(* IEC 61131-3 sources: HappyLearnCodesys/content/softmotion/Robotics_PickAndPlace, 6 files *)

(* ---- GVL.st ---- *)
(*
    檔案用途：定義本範例中三角機器人、輸送帶與旋轉工作台的幾何位置常數，
              以及用來切換「自動／手動放環」的全域旗標。
    教學重點：這些數值會直接影響實際運動軌跡與畫面位置，修改前請先對照
              `DeviceTree_Axes.md` 與各 POU 程式中的使用方式再調整。
*)
VAR_GLOBAL CONSTANT
    gcTripodTransX : LREAL := 0;       // Tripod 機構在世界座標中的 X 平移量
    gcTripodTransY : LREAL := 0;       // Tripod 機構在世界座標中的 Y 平移量
    gcTripodTransZ : LREAL := 1700;    // Tripod 機構在世界座標中的 Z 平移量（機器人高度）

    gcTripodSize : LREAL := 180;       // Tripod 幾何尺寸基準，影響工作空間與 TCP 半徑

    gcBeltTransX : LREAL := 0;         // 輸送帶座標系（PCS_2）在世界座標中的 X 位置
    gcBeltTransY : LREAL := 500;       // 輸送帶座標系在世界座標中的 Y 位置
    gcBeltTransZ : LREAL := 0;         // 輸送帶座標系在世界座標中的 Z 位置

    gcTableTransX : LREAL := 0;        // 旋轉工作台座標系（PCS_1）在世界座標中的 X 位置
    gcTableTransY : LREAL := -500;     // 旋轉工作台座標系在世界座標中的 Y 位置
    gcTableTransZ : LREAL := 0;        // 旋轉工作台座標系在世界座標中的 Z 位置

    gcTCP_Ring : LREAL := 0.02 * gcTripodSize + 15;   // 末端工具座標系到圓環下緣的距離

    gcTripod1PosOrig : LREAL := 50;    // Tripod1 初始軸位置
    gcTripod2PosOrig : LREAL := 75;    // Tripod2 初始軸位置
    gcTripod3PosOrig : LREAL := 25;    // Tripod3 初始軸位置
END_VAR
VAR_GLOBAL
    gbSetRing : BOOL;                  // TRUE：由操作者手動要求在轉盤上放一個新環
    gbAutomatic : BOOL := TRUE;        // TRUE：環依邏輯自動連續產生；FALSE：完全由 gbSetRing 控制
END_VAR

(* ---- Cone.st ---- *)
(*
    檔案用途：
      以狀態機方式描述單一圓錐（Cone）在輸送帶上的一生：
      何時出現、如何被輸送帶帶動、何時離開工作區域，以及如何更新 PCS_2。
    教學重點：
      - 透過 MC_TrackConveyorBelt 追蹤輸送帶上的物件位置，並與 Tripod 軸組連動。
      - 觀察 REPEAT / UNTIL 與 state / stateOld 的組合，如何實作「直到狀態穩定」的迴圈。
      - 理解 pActiveCone 與 pPreviousCone 指標，如何在三顆圓錐之間接續產生與移動。
*)
FUNCTION_BLOCK Cone
VAR_IN_OUT
	pActiveCone : POINTER TO Cone;
END_VAR
VAR_INPUT
	pPreviousCone : POINTER TO Cone;
END_VAR
VAR_OUTPUT
	pos : MC_COORD_REF;
	state : DINT;
	bOnBelt : BOOL;
END_VAR
VAR
	conveyorBeltOrigin : MC_COORD_REF := (X := gcBeltTransX, Y := gcBeltTransY, Z := gcBeltTransZ);
	initialConePosition : MC_COORD_REF := (X := -925, Z := 125);
	tcb : MC_TrackConveyorBelt := (ConveyorBeltOrigin := conveyorBeltOrigin,
								   InitialObjectPosition := initialConePosition,
								   CoordSystem := SMC_COORD_SYSTEM.PCS_2);
	f : SMC_Frame;
	stateOld : DINT;
END_VAR

REPEAT
	stateOld := state;
	CASE state OF
	0:	//cone invisible
		IF NOT Robot.bDontChangePCS_2 THEN
			IF pPreviousCone^.bOnBelt AND pPreviousCone^.pos.X >= -250 THEN
				tcb(Execute := FALSE, AxisGroup := Tripod, ConveyorBelt := DriveConveyorBelt);
				tcb.Execute := TRUE;
				state := state + 10;
			END_IF
		END_IF
	10:	//linking PCS_2 to the position of the cone
		IF tcb.Done THEN
			bOnBelt := TRUE;
			pActiveCone := THIS;
			state := state + 10;
		END_IF
	20:	//cone on belt
		tcb.cs.GetPose(cs := f, fTime := Tripod1.fTaskCycle);
		SMC_Frame_To_CoordRef(c := pos, f := f);
		IF pos.X >= gcBeltTransX + 725 THEN
			bOnBelt := FALSE;
			state := 0;
		END_IF
	END_CASE
	tcb(AxisGroup := Tripod, ConveyorBelt := DriveConveyorBelt);
UNTIL state = stateOld
END_REPEAT

(* ---- Ring.st ---- *)
(*
    檔案用途：
      以狀態機方式描述單一圓環（Ring）從轉盤待命、被機器人取走、
      一直到被放到圓錐上、再回到初始狀態的整個流程。
    教學重點：
      - 使用 MC_TrackRotaryTable 取得轉盤上物件的即時位置，並映射到 PCS_1。
      - 觀察如何根據 Robot 的輸出旗標（bReadyForMotion、bRingAttached、pTargetCone）
        來協調「轉盤上兩個圓環」與「機器人」之間的合作。
      - 練習閱讀以 DINT state 切分的多段狀態（0/10/20/30/40/50），對照實際動作想像流程。
*)
FUNCTION_BLOCK Ring
VAR_INPUT
	pOtherRing : POINTER TO Ring;
	startPos : MC_COORD_REF;
END_VAR
VAR_OUTPUT
	pos : MC_COORD_REF;
	state : DINT;
	bOnTable : BOOL;
END_VAR
VAR
	stateOld : DINT;
	fTemp : LREAL;
	f : SMC_Frame;
	rotaryTableOrigin : MC_COORD_REF := (X := gcTableTransX, Y := gcTableTransY, Z := gcTableTransZ);
	initialObjectPosition : MC_COORD_REF := (Y := 400, Z := 20 + 10);
	trt : MC_TrackRotaryTable := (RotaryTableOrigin := rotaryTableOrigin, initialObjectPosition := initialObjectPosition, CoordSystem := SMC_COORD_SYSTEM.PCS_1);
	pCone : POINTER TO Cone;
END_VAR

REPEAT
	stateOld := state;
	CASE state OF
	0:	//ring at original position
		pos := startPos;
		IF Robot.bReadyForMotion AND
		   (pOtherRing^.state = 0 OR pOtherRing^.state >= 40) AND
		   (gbSetRing OR gbAutomatic) THEN
			trt(Execute := FALSE, AxisGroup := Tripod, RotaryTable := DriveRotaryTable);
			trt.Execute := TRUE;
			state := state + 10;
		END_IF

	10:	//linking PCS_1 to the position of the ring
		IF trt.Done THEN
			state := state + 10;
		END_IF

	20:	//ring on rotary-table, wait until robot is free
		trt.cs.GetPose(cs := f, fTime := Tripod1.fTaskCycle);
		SMC_Frame_To_CoordRef(c := pos, f := f);
		IF NOT Robot.bRingAttached THEN
			state := state + 10;
		END_IF

	30: //waiting for takeoff
		trt.cs.GetPose(cs := f, fTime := Tripod1.fTaskCycle);
		SMC_Frame_To_CoordRef(c := pos, f := f);
		IF Robot.bRingAttached THEN
			state := state + 10;
		END_IF

	40:	//ring attached to robot
		pos.X := Robot.readPos.Position.c.X;
		pos.Y := Robot.readPos.Position.c.Y;
		pos.Z := Robot.readPos.Position.c.Z - gcTCP_Ring;
		IF NOT Robot.bRingAttached THEN
			pCone := Robot.pTargetCone;
			state := state + 10;
		END_IF

	50:	//ring placed on cone
		pos.X := pCone^.pos.X;
		pos.Y := pCone^.pos.Y;
		pos.Z := pCone^.pos.Z;
		IF NOT pCone^.bOnBelt THEN
			state := 0;
		END_IF
	END_CASE

	trt(AxisGroup := Tripod, RotaryTable := DriveRotaryTable);
UNTIL state = stateOld
END_REPEAT

bOnTable := state = 20 OR state = 30;

(* ---- DepictorCalculations.st ---- *)
(*
    檔案用途：
      計算用於可視化的標記座標陣列 aafPos，讓視覺介面能畫出輸送帶路徑
      以及 Tripod 運動軌跡的參考線。
    教學重點：
      - 透過 Tripod_Lin_Depictor 取得 Tripod 軸組的線性插補資訊，作為可視化基底。
      - 使用 SIN、COS 與多段 if/else 邏輯，組合出一條封閉的輸送帶路徑。
      - 練習將實際軸位置（DriveConveyorBelt.fSetPosition 等）轉換成畫面上的座標點。
*)
PROGRAM DepictorCalculations
VAR_OUTPUT
	aafPos : ARRAY[0..9] OF ARRAY[0..1] OF LREAL;
END_VAR
VAR
	dep : Tripod_Lin_Depictor;
	fTemp : LREAL;
	i : INT;
END_VAR

//tripod
IF Robot.state >= 40 THEN
	dep(group := Tripod, kin := Tripod.trafo);
END_IF

//markings on belt
FOR i := 0 TO 9 DO
	fTemp := DriveConveyorBelt.fSetPosition + INT_TO_LREAL(i) / 10 * DriveConveyorBelt.fPositionPeriod;
	IF fTemp >= DriveConveyorBelt.fPositionPeriod THEN
		fTemp := fTemp - DriveConveyorBelt.fPositionPeriod;
	END_IF

	IF fTemp <= 1000 THEN
		aafPos[i][0] := fTemp;
		aafPos[i][1] := 50;
	ELSE
		fTemp := fTemp - 1000;
		IF fTemp < 50 * SMC_PI THEN
			aafPos[i][0] := 1000 + 50 * SIN(fTemp / 50);
			aafPos[i][1] := 50 * COS(fTemp / 50);
		ELSE
			fTemp := fTemp - 50 * SMC_PI;
			IF fTemp <= 2000 THEN
				aafPos[i][0] := 1000 - fTemp;
				aafPos[i][1] := -50;
			ELSE
				fTemp := fTemp - 2000;
				IF fTemp < 50 * SMC_PI THEN
					aafPos[i][0] := -1000 - 50 * SIN(fTemp / 50);
					aafPos[i][1] := -50 * COS(fTemp / 50);
				ELSE
					fTemp := fTemp - 50 * SMC_PI;
					aafPos[i][0] := -1000 + fTemp;
					aafPos[i][1] := 50;
				END_IF
			END_IF
		END_IF
	END_IF
END_FOR

(* ---- Environment.st ---- *)
(*
    檔案用途：
      負責「環境」相關的裝置控制，包括旋轉工作台與輸送帶的驅動，
      並管理所有圓錐（Cone）與圓環（Ring）的狀態機，提供給機器人程式使用。
    教學重點：
      - 將與機器人本體無關、但會影響工作流程的設備集中在一支 PROGRAM 中管理。
      - 觀察如何透過 FUNCTION_BLOCK 實例（Cone、Ring）與指標，建立物件之間的關聯。
      - 使用簡單的初始化旗標 bInit 來區分「第一次循環」與「正常運轉」的寫法。
*)
PROGRAM Environment
VAR_OUTPUT
	cone1, cone2, cone3 : Cone;
	ring1, ring2 : Ring;
	bRingOnTable : BOOL;
	pActiveCone : POINTER TO Cone;	//the cone corresponding to PCS_2
END_VAR
VAR
	powRotaryTable : MC_Power := (Enable := TRUE, bRegulatorOn := TRUE, bDriveStart := TRUE);
	powConveyorBelt : MC_Power := (Enable := TRUE, bRegulatorOn := TRUE, bDriveStart := TRUE);
	mvRotaryTable : MC_MoveVelocity := (Execute := TRUE, Velocity := 50, Acceleration := 30, Deceleration := 30, Jerk := 1000);
	mvConveyorBelt : MC_MoveVelocity := (Execute := TRUE, Velocity := 300, Acceleration := 150, Deceleration := 150, Jerk := 1000);

	ring1StartPos : MC_COORD_REF := (X := 75, Y := 100, Z := 0);
	ring2StartPos : MC_COORD_REF := (X := -75, Y := 100, Z := 0);
	bInit : BOOL := TRUE;
END_VAR

//moving rotary-table-/ conveyor-belt-drive
powRotaryTable(Axis := DriveRotaryTable);
powConveyorBelt(Axis := DriveConveyorBelt);
IF NOT (powRotaryTable.Status AND powConveyorBelt.Status) THEN
	RETURN;
END_IF
mvRotaryTable(Axis := DriveRotaryTable);
mvConveyorBelt(Axis := DriveConveyorBelt);

//state-machines of cones / handling of PCS_2
IF bInit THEN
	cone1.Start();
END_IF
cone1(pActiveCone := pActiveCone, pPreviousCone := ADR(cone3));
cone2(pActiveCone := pActiveCone, pPreviousCone := ADR(cone1));
cone3(pActiveCone := pActiveCone, pPreviousCone := ADR(cone2));

//state-machines of rings / handling of PCS_1
IF bInit THEN
	ring1.startPos := ring1StartPos;
	ring2.startPos := ring2StartPos;
END_IF
ring1(pOtherRing := ADR(ring2));
ring2(pOtherRing := ADR(ring1));
bRingOnTable := ring1.bOnTable OR ring2.bOnTable;

bInit := FALSE;

(* ---- Robot.st ---- *)
(*
    檔案用途：
      控制 Tripod 三角機器人完成「從旋轉工作台拾取圓環，放置到輸送帶上圓錐」的
      完整 Pick & Place 循環，並回報目前是否可動作與是否已夾持圓環。
    教學重點：
      - 觀察如何使用多顆 MC_Power、MC_SetPosition、MC_MoveLinear* 等運動控制 FB
        來建立啟動流程與多段直線軌跡。
      - 搭配座標系（WCS、PCS_1、PCS_2）與位置常數，理解不同工位之間的轉換。
      - 透過整數變數 state 所構成的狀態機，練習閱讀與設計順序控制流程。
*)
PROGRAM Robot
VAR_OUTPUT
    bReadyForMotion : BOOL;
	bRingAttached : BOOL;
	bDontChangePCS_2 : BOOL;	//there are several commands using PCS_2, which shall not change in the meantime
	pTargetCone : POINTER TO Cone;
END_VAR
VAR
    pwA1 : MC_Power := (Enable:= TRUE, bRegulatorOn:= TRUE, bDriveStart:= TRUE);
    pwA2 : MC_Power := (Enable:= TRUE, bRegulatorOn:= TRUE, bDriveStart:= TRUE);
    pwA3 : MC_Power := (Enable:= TRUE, bRegulatorOn:= TRUE, bDriveStart:= TRUE);
    spA1, spA2, spA3 : MC_SetPosition;

	enable : MC_GroupEnable;
	setCoord : MC_SetCoordinateTransform;
    mcs : MC_COORD_REF;

    mvToRing : MC_MoveLinearAbsolute := (Velocity := VEL, Acceleration := ACC, Deceleration := ACC, Jerk := JRK, Name:= 'Move to ring');
	mvToRestPos : MC_MoveLinearAbsolute := (Velocity := VEL, Acceleration := ACC, Deceleration := ACC, Jerk := JRK, Name:= 'Move to rest position');
	mvAboveCone : MC_MoveLinearAbsolute := (Velocity := VEL, Acceleration := ACC, Deceleration := ACC, Jerk := JRK, Name:= 'Move above cone');
	mvUpFromRing : MC_MoveLinearRelative := (Velocity := VEL, Acceleration := ACC, Deceleration := ACC, Jerk := JRK, Name:= 'Move up from ring');

	mvDownToCone : MC_MoveLinearAbsolute := (Velocity := VEL, Acceleration := ACC, Deceleration := ACC, Jerk := JRK, Name:= 'Move down to cone');
	mvUpFromCone : MC_MoveLinearAbsolute := (Velocity := VEL, Acceleration := ACC, Deceleration := ACC, Jerk := JRK, Name:= 'Move up from cone');

    mvBack : MC_MoveLinearAbsolute := (Velocity := VEL, Acceleration := ACC, Deceleration := ACC, Jerk := JRK, Name:= 'Move back');

	readStatus : MC_GroupReadStatus;
    readPos : MC_GroupReadActualPosition;

	state : INT;
	ton : TON := (PT := T#200MS);
END_VAR
VAR CONSTANT
    VEL : LREAL :=   1000 ;
    ACC : LREAL :=  10000 ;
    JRK : LREAL := 100000 ;

    POS_ABOVE_RING_PCS_1 : SMC_POS_REF := (c:= (X:= 0, Y:= 0, Z:= gcTCP_Ring)) ;
    POS_ABOVE_CONE_PCS_2 : SMC_POS_REF := (c:= (X:= 0, Y:= 0, Z:= 200)) ;
    POS_ON_CONE_PCS_2 : SMC_POS_REF := (c:= (X:= 0, Y:= 0, Z:= gcTCP_Ring)) ;
    POS_REST_WCS : SMC_POS_REF := (c:= (X:= 0, Y:= 0, Z:= 300)) ;
END_VAR

pwA1(Axis:= Tripod1);
pwA2(Axis:= Tripod2);
pwA3(Axis:= Tripod3);

CASE state OF
0:
    IF pwA1.Status AND pwA2.Status AND pwA3.Status THEN
        state := state + 10;
	END_IF

10:	//starting at given axis-positions
    spA1(Axis:= Tripod1, Execute:= TRUE, Position:= gcTripod1PosOrig);
    spA2(Axis:= Tripod2, Execute:= TRUE, Position:= gcTripod2PosOrig);
    spA3(Axis:= Tripod3, Execute:= TRUE, Position:= gcTripod3PosOrig);

    IF spA1.Done AND spA2.Done AND spA3.Done THEN
		setCoord(AxisGroup := Tripod, Execute := FALSE);
        state := state + 10;
	END_IF

20:	//telling the robot its position in space
	mcs.X := gcTripodTransX;
	mcs.Y := gcTripodTransY;
	mcs.Z := gcTripodTransZ;
    setCoord(
	        AxisGroup := Tripod,
            Execute := TRUE,
            CoordTransform := mcs,
            CoordSystem := SMC_COORD_SYSTEM.MCS);

    IF setCoord.Done THEN
        state := state + 10;
	END_IF

30: //enabling the axis group
    enable(AxisGroup:= Tripod, Execute:= TRUE);
    IF enable.Done THEN
		state := state + 10;
    END_IF

40:
	IF Environment.bRingOnTable THEN
		//approaching a ring on the table
		mvToRing(AxisGroup:= Tripod, Execute := FALSE);
		mvToRing.Position := POS_ABOVE_RING_PCS_1 ;
		mvToRing.BufferMode := MC_BUFFER_MODE.BlendingHigh;
		mvToRing.TransitionMode := MC_TRANSITION_MODE.TMCornerDistance;
		mvToRing.TransitionParameter[0] := 500;
		mvToRing.CoordSystem := SMC_COORD_SYSTEM.PCS_1;
		mvToRing.Execute := TRUE;
    	state := state + 10;
	END_IF

50:
    IF mvToRing.Done THEN
		ton(IN := FALSE);
		state := state + 10;
	END_IF

60:
	ton(IN := TRUE);
	//waiting some time (following the ring)
	IF ton.Q THEN
		//moving upwards (still in PCS_1)
		mvUpFromRing(AxisGroup:= Tripod, Execute := FALSE);
		mvUpFromRing.Distance.c.Z := 150;
		mvUpFromRing.CoordSystem := SMC_COORD_SYSTEM.PCS_1;
		mvUpFromRing.BufferMode := MC_BUFFER_MODE.Buffered;
		mvUpFromRing.TransitionMode := MC_TRANSITION_MODE.TMNone;
		mvUpFromRing.Execute := TRUE;
		state := state + 10;
	END_IF

70:
	IF mvUpFromRing.CommandAccepted THEN
		//neutral position
		mvToRestPos(AxisGroup:= Tripod, Execute := FALSE);
		mvToRestPos.Position := POS_REST_WCS ;
		mvToRestPos.CoordSystem := SMC_COORD_SYSTEM.WCS;
		mvToRestPos.BufferMode := MC_BUFFER_MODE.BlendingHigh;
		mvToRestPos.TransitionMode := MC_TRANSITION_MODE.TMCornerDistance;
		mvToRestPos.TransitionParameter[0] := 500 ;
		mvToRestPos.Execute := TRUE;
		state := state + 10;
	END_IF

80:
	IF mvToRestPos.CommandAccepted THEN
		//moving to some position above the next cone
		pTargetCone := Environment.pActiveCone;
		mvAboveCone(AxisGroup:= Tripod, Execute := FALSE);
		mvAboveCone.Position := POS_ABOVE_CONE_PCS_2 ;
		mvAboveCone.CoordSystem := SMC_COORD_SYSTEM.PCS_2;
		mvAboveCone.BufferMode := MC_BUFFER_MODE.BlendingHigh;
		mvAboveCone.TransitionMode := MC_TRANSITION_MODE.TMCornerDistance;
        mvAboveCone.TransitionParameter[0] := 1000 ;
		mvAboveCone.Execute := TRUE;
		state := state + 10;
	END_IF

90:
	IF mvAboveCone.CommandAccepted THEN
		//approaching the cone
		mvDownToCone(AxisGroup:= Tripod, Execute := FALSE);
		mvDownToCone.Position := POS_ON_CONE_PCS_2 ;
		mvDownToCone.BufferMode := MC_BUFFER_MODE.BlendingHigh;
		mvDownToCone.TransitionMode := MC_TRANSITION_MODE.TMCornerDistance;
		mvDownToCone.CoordSystem := SMC_COORD_SYSTEM.PCS_2;
		mvDownToCone.TransitionParameter[0] := 500;
		mvDownToCone.Execute := TRUE;
		state := state + 10;
	END_IF

100:
	IF mvDownToCone.Done THEN
		//moving upwards (still following the belt)
		mvUpFromCone(AxisGroup:= Tripod, Execute := FALSE);
		mvUpFromCone.Position := POS_ABOVE_CONE_PCS_2 ;
		mvUpFromCone.BufferMode := MC_BUFFER_MODE.Buffered;
		mvUpFromCone.TransitionMode := MC_TRANSITION_MODE.TMNone;
		mvUpFromCone.CoordSystem := SMC_COORD_SYSTEM.PCS_2;
		mvUpFromCone.Execute := TRUE;
		state := state + 10;
	END_IF

110:
	IF mvUpFromCone.CommandAccepted THEN
		//moving back
		mvBack(AxisGroup:= Tripod, Execute := FALSE);
		mvBack.Position := POS_REST_WCS ;
		mvBack.CoordSystem := SMC_COORD_SYSTEM.WCS;
		mvBack.BufferMode := MC_BUFFER_MODE.BlendingHigh;
		mvBack.TransitionMode := MC_TRANSITION_MODE.TMCornerDistance;
		mvBack.TransitionParameter[0] := 500;
		mvBack.Execute := TRUE;
		state := state + 10;
	END_IF

120:
	IF mvBack.CommandAccepted THEN
		state := 40;
	END_IF

END_CASE

mvToRing(AxisGroup := Tripod);
mvUpFromRing(AxisGroup := Tripod);
mvToRestPos(AxisGroup := Tripod);
mvAboveCone(AxisGroup := Tripod);
mvDownToCone(AxisGroup := Tripod);
mvUpFromCone(AxisGroup := Tripod);
mvBack(AxisGroup := Tripod);

readStatus(AxisGroup := Tripod, Enable := TRUE);
readpos(AxisGroup:= Tripod, Enable:= TRUE, CoordSystem:= SMC_COORD_SYSTEM.WCS);

bReadyForMotion := NOT readStatus.GroupDisabled AND NOT readStatus.GroupErrorStop;
bRingAttached := state >= 70 AND state <= 100;
bDontChangePCS_2 := state >= 90 AND state <= 110;
